{attribute 'qualified_only'}
{attribute 'strict'}
TYPE E_TestState :
(
	IDLE,
	EQ2HOR,
	HOR2EQ,
	EQ2EQ,
	JD2LST,
	ERROR
);
END_TYPE

(* stored: Version 1.1.0.1, ProductVersion 3.1.4024.12
   DUT E_TestState: Id {7e890740-17ec-420f-b803-923d73845ddd} *)
